FUNCTION_BLOCK FB_Betriebsarten
VAR_INPUT
	bIAnlageEin:			BOOL;		// Taster Anlage eingeschaltet
	bISAnlageAus: 			BOOL;		// Taster Anlage ausgeschaltet
	bIManAuto:				BOOL;		// Schalter Manuell / Automatik
	bINotAus:				BOOL;		// Not-Aus, 1 = i.O, 0 = betätigt
	bIDauerEinzel:			BOOL;		// Schalter Dauer- bzw. Einzelbetrieb, 0 = Dauer, 1 = Einzelbetrieb
	bIStart:				BOOL;		// Starttaster 
END_VAR
VAR_OUTPUT
	bOAnlageEin:			BOOL;		// 1 = Anlage eingeschaltet
	bOManuell:				BOOL;		// 1 = Anlage Manuellbetrieb
	bOAuto:					BOOL;		// 1 = Anlage im Autobetrieb
	bOEinzelZyklus:			BOOL;		// 1 = Einzelzyklus aktiv
	bODauerZyklus:			BOOL;		// 1 = Dauerzyklus aktiv
	bOStoerung:				BOOL;		// 1 = Stoerung vorhanden (Not-Aus)
	bOImpEinzelSchritt:		BOOL;		// Impuls bei Einzelschrittbetrieb von Start-Taster
	bOImpDauerZyklus:		BOOL;		// Impuls bei Dauerschrittbetrieb von Start-Taster
	stAnlagenzustand:		ST_Anlagenzustand;
END_VAR
VAR_IN_OUT
END_VAR
VAR
	bSVAnlageEin:			BOOL;		// Variable 1 = Anlage eingeschaltet 
	lastbEinzelImp: 		BOOL;		// Letzter Zustand Tipp-Impuls für Flankenerkennung
	lastbDauerImp: 			BOOL;		// Letzter Zustand Dauer-Impuls für Flankenerkennung
END_VAR

(*
- Wenn Not-Aus aktiv, alle FB-Ausgänge rücksetzen und Ausgang vqx_Störung setzen 
- vqx_AnlageEin speichernd set/reset mit vix_AnlageEin und vix_AnlageAus (Öffner) 
- Wenn Anlage nicht eigeschaltet, dann alle Ausgänge rücksetzen 
- vqx_Man wird gesetzt, wenn vix_ManAuto auf Man (False) steht und Anlage eingeschaltet ist 
- vqx_Auto wird gesetzt, wenn vix_ManAuto auf Auto (True) steht und Anlage eingeschaltet ist 
- vqx_EinzZykl wird gesetzt, wenn vix_DauerEinz auf Einzel (True) steht und die Anlage eingeschaltet ist 
- vqx_ImpEinzelSchritt wird für 1 Zyklus logisch "1" wenn der Einzel-Zyklus aktiv ist und die Anlage eingeschaltet ist und der Start-Taster gedrückt wird. 
- vqx_DauerZykl wird gesetzt, wenn vix_DauerEinz auf Dauer (False) steht und der Automatikbetrieb aktiv und die Anlage eingeschaltet ist 
- vqx_ImpDauerZykl wird für 1 Zyklus logisch "1" wenn Dauer-Zyklus aktiv ist und die Anlage eingeschaltet ist und der Start-Taster gedrückt wird.
*)

// IF bIStart THEN
// 	stAnlagenzustand.bAnlageEin := TRUE;
// END_IF

IF bINotAus THEN
bOAnlageEin				:= FALSE;
bOManuell				:= FALSE;
bOAuto					:= FALSE;
bOEinzelZyklus			:= FALSE;		
bODauerZyklus			:= FALSE;
bOImpEinzelSchritt		:= FALSE;		
bOImpDauerZyklus		:= FALSE;
bOStoerung				:= TRUE;
END_IF

END_FUNCTION_BLOCK

(* stored: Version 1.1.0.1
   POU FB_Betriebsarten: Id {9f3c47b0-eea8-486d-bc24-1b316794b68c}, SpecialFunc None *)
